FUNCTION_BLOCK GenericCylinderModelType2 (* Composite Function Block Type *)
  (* Standard: 61499-2 *)
  (* Version 0.0, 2/3/2012, XPMUser, nxtControl GmbH, template *)
  PACKAGE Main;
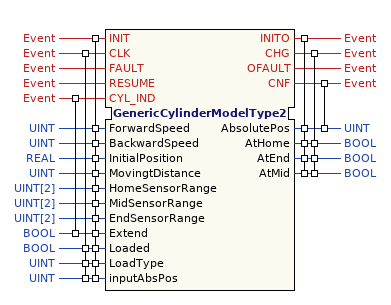
  EVENT_INPUT
    INIT WITH ForwardSpeed, BackwardSpeed, Extend, HomeSensorRange, EndSensorRange, InitialPosition, LoadType, MovingtDistance, Loaded, MidSensorRange, inputAbsPos; (* Initialization Request *)
    CLK WITH LoadType, Loaded, inputAbsPos; (* Clock signal *)
    FAULT;
    RESUME;
    CYL_IND WITH Extend;
  END_EVENT
  EVENT_OUTPUT
    INITO WITH AbsolutePos, AtHome, AtEnd, AtMid; (* Initialization Confirm *)
    CHG WITH AtEnd, AtHome, AtMid; (* Indicate data outputs changed *)
    OFAULT;
    CNF WITH AbsolutePos;
  END_EVENT
  VAR_INPUT
    ForwardSpeed : UINT; (* Forward speed *)
    BackwardSpeed : UINT; (* Backward speed *)
    InitialPosition : REAL; (* Initial position *)
    MovingtDistance : UINT; (* Moving distance *)
    HomeSensorRange : ARRAY [0..1] OF UINT; (* Detection range of home sensor *)
    MidSensorRange : ARRAY [0..1] OF UINT; (* Detection range of home sensor *)
    EndSensorRange : ARRAY [0..1] OF UINT; (* Detection range of end sensor *)
    Extend : BOOL;
    Loaded : BOOL;
    LoadType : UINT;
    inputAbsPos : UINT;
  END_VAR
  VAR_OUTPUT
    AbsolutePos : UINT; (* Current position *)
    AtHome : BOOL; (* Detected at home position *)
    AtEnd : BOOL; (* Detected at end position *)
    AtMid : BOOL;
  END_VAR
  FBS
    Home : RangeSensor;
    Middle : RangeSensor;
    End : RangeSensor;
    FB1 : MovingStatusType2;
    Position : LinearMotionLoad;
  END_FBS
  EVENT_CONNECTIONS
    Position.INITO TO Home.INIT;
    Home.INITO TO Middle.INIT;
    Middle.INITO TO End.INIT;
    End.INITO TO INITO;
    Home.CHG TO CHG;
    End.CHG TO CHG;
    Middle.CHG TO CHG;
    Position.CHG TO CNF;
    CLK TO Position.CLK;
    Position.CHG TO Home.CLK;
    Position.CHG TO Middle.CLK;
    Position.CHG TO End.CLK;
    INIT TO FB1.INIT;
    CYL_IND TO FB1.CLK;
    FAULT TO FB1.FAULT;
    RESUME TO FB1.RESUME;
    FB1.INITO TO Position.INIT;
    FB1.OFAULT TO OFAULT;
  END_CONNECTIONS
  DATA_CONNECTIONS
    Loaded TO Position.Loaded;
    LoadType TO Position.LoadType;
    EndSensorRange TO End.Zone;
    HomeSensorRange TO Home.Zone;
    Position.RelativePos TO Middle.Position;
    Position.RelativePos TO End.Position;
    Home.Detected TO AtHome;
    Middle.Detected TO AtMid;
    End.Detected TO AtEnd;
    ForwardSpeed TO Position.ForwardSpeed;
    BackwardSpeed TO Position.BackwardSpeed;
    InitialPosition TO Position.InitialPosition;
    MovingtDistance TO Position.MovingDistance;
    Position.AbsolutePos TO AbsolutePos;
    Position.RelativePos TO Home.Position;
    MidSensorRange TO Middle.Zone;
    Extend TO FB1.Extend;
    inputAbsPos TO Position.inputAbsPos;
    FB1.C_FWD TO Position.MoveForwards;
    FB1.C_BWD TO Position.MoveBackwards;
  END_CONNECTIONS
END_FUNCTION_BLOCK
